PROGRAM POU
VAR
	Ton1 :ton;
	Ton2 :ton;
	
END_VAR


ton1(PT := T#2S);
ton2(PT := T#2S);


IF ton2.Q = TRUE THEN
			ton1.in :=FALSE;
			ton2.IN :=FALSE;
			
ELSIF ton1.Q = TRUE THEN
		ton2.IN := TRUE;
				
ELSIF ton2.Q = FALSE THEN
	ton1.IN := TRUE;
	
	
END_IF

END_PROGRAM

(* stored: Version 1.1.0.1, ProductVersion 3.1.4024.12
   POU POU: Id {250b1260-1cee-43b3-87a3-fd773fbfbb19}, SpecialFunc None *)
